ABB RobotStudio station: estacion_lab1_nike_plano.rsstn

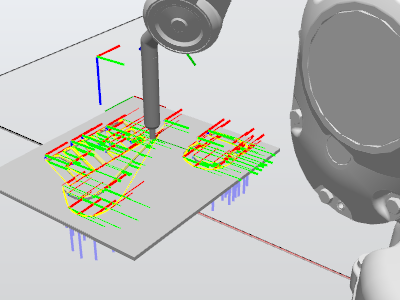
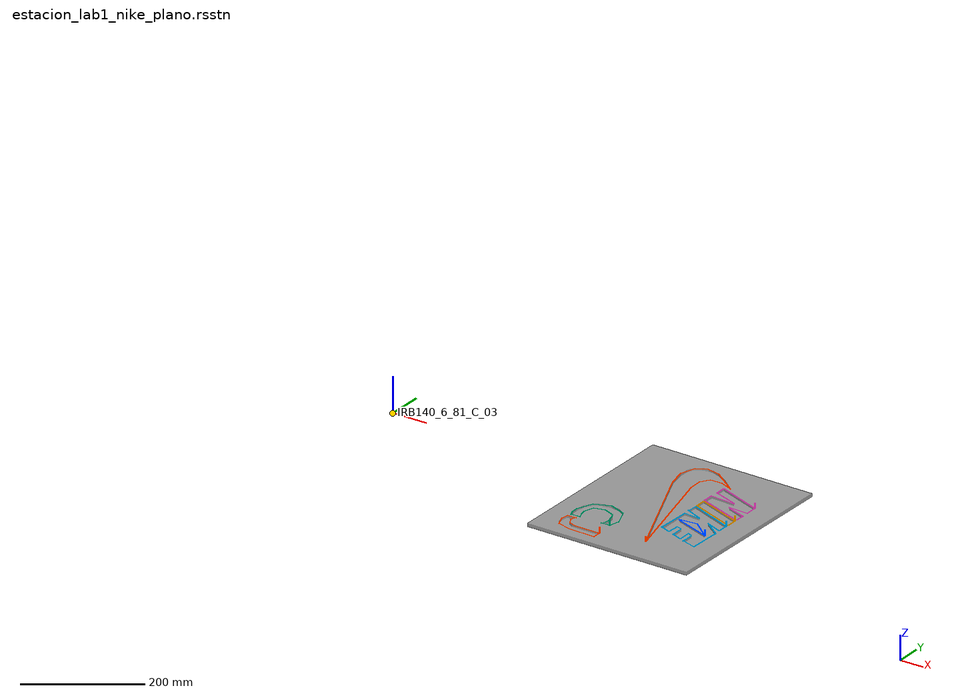
[picture v1: parts stored in the station drawn from their meshes, with robot base, taught points and paths (robot models come from the ABB library and are not in the file)]
Station estacion_lab1_nike_plano (saved by RobotStudio 24.1.10693.0)
Controller ControladorLab1
  mechanical unit ROB_1: IRB140_6_81_C_03, 6 joints, base frame (0, 0, 0) mm
Layout (positions relative to the parent item):
  - IRB140_6_81_C_03 [mechanism, from %ABB.RobotStudio.Models.IRB140%\IRB140_6_81_C_G_03.rslib] at (0, 0, 0) mm; joint values [-0.2293, 0.8636, 0.1936, 2.4826, 0.316, 2.0103] (rad or m)
  - Silueta_nike_nombres [part] at (550, 0, 0) mm, rotated rx 0 ry 0 rz -90 deg, size 349.5 x 310.3 x 6 mm
  - ToolLab1 [mechanism] at (562.41, -118.55, 208.97) mm, rotated rx -135 ry 0 rz -87.52 deg
      TCP ToolLab1 at (0.11, 120.32, 166.73) mm, rotated rx -45 ry 0 rz 0 deg
      links: HerramientaMarcadorEnsamblada v1
Attachment: ToolLab1 is attached to IRB140_6_81_C_03 / Link6
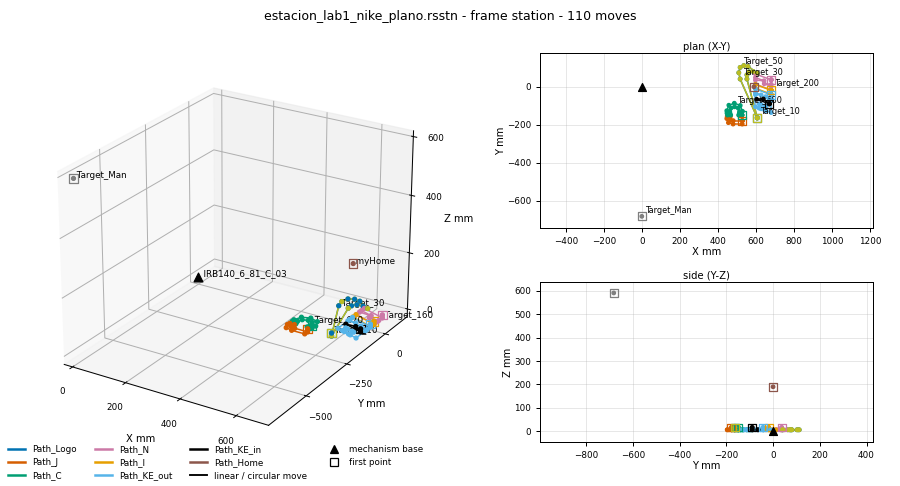
[picture p0: tool path of estacion_lab1_nike_plano.rsstn in frame station, 110 of 110 moves have a stored position in this frame; points joined in program order, loops and branches not executed]
Targets, tools, work objects and paths stored in the station, written as RAPID:
! task T_ROB1
MODULE CalibData
  PERS tooldata ToolLab1:=[TRUE,[[0.111,120.323,166.727],[0.923879533,-0.382683432,0,0]],[1,[0,0,1],[1,0,0,0],0,0,0]];
  TASK PERS wobjdata Workobject_1:=[FALSE,TRUE,"",[[722.891,-215.257,6],[0,0,1,0]],[[0,0,0],[1,0,0,0]]];
ENDMODULE

! task T_ROB1
MODULE Module1
  CONST robtarget Target_10:=[[115.3493902,51.778117998,-10],[0.69165817,0,0,-0.722225017],[0,0,0,0],[9E+09,9E+09,9E+09,9E+09,9E+09,9E+09]];
  CONST robtarget Target_20:=[[115.3493902,51.778117998,0],[0.69165817,0,0,-0.722225017],[0,0,0,0],[9E+09,9E+09,9E+09,9E+09,9E+09,9E+09]];
  CONST robtarget Target_30:=[[205.483730587,256.22918847,0],[0.69165817,0,0,-0.722225017],[0,0,0,0],[9E+09,9E+09,9E+09,9E+09,9E+09,9E+09]];
  CONST robtarget Target_40:=[[212.583843163,289.281706109,0],[0.69165817,0,0,-0.722225017],[0,0,0,0],[9E+09,9E+09,9E+09,9E+09,9E+09,9E+09]];
  CONST robtarget Target_50:=[[205.483730587,317.417949705,0],[0.69165817,0,0,-0.722225017],[0,0,0,0],[9E+09,9E+09,9E+09,9E+09,9E+09,9E+09]];
  CONST robtarget Target_60:=[[186.065561002,327.253449307,0],[0.69165817,0,0,-0.722225017],[0,0,0,0],[9E+09,9E+09,9E+09,9E+09,9E+09,9E+09]];
  CONST robtarget Target_70:=[[164.044058996,322.576768388,0],[0.69165817,0,0,-0.722225017],[0,0,0,0],[9E+09,9E+09,9E+09,9E+09,9E+09,9E+09]];
  CONST robtarget Target_80:=[[115.3493902,287.739568507,0],[0.69165817,0,0,-0.722225017],[0,0,0,0],[9E+09,9E+09,9E+09,9E+09,9E+09,9E+09]];
  CONST robtarget Target_90:=[[137.113893268,295.786272701,0],[0.69165817,0,0,-0.722225017],[0,0,0,0],[9E+09,9E+09,9E+09,9E+09,9E+09,9E+09]];
  CONST robtarget Target_100:=[[159.309752186,294.100202202,0],[0.69165817,0,0,-0.722225017],[0,0,0,0],[9E+09,9E+09,9E+09,9E+09,9E+09,9E+09]];
  CONST robtarget Target_110:=[[169.98114276,278.010063881,0],[0.69165817,0,0,-0.722225017],[0,0,0,0],[9E+09,9E+09,9E+09,9E+09,9E+09,9E+09]];
  CONST robtarget Target_120:=[[169.942954093,256.22918847,0],[0.69165817,0,0,-0.722225017],[0,0,0,0],[9E+09,9E+09,9E+09,9E+09,9E+09,9E+09]];
  CONST robtarget Target_130:=[[115.3493902,51.778117998,0],[0.69165817,0,0,-0.722225017],[0,0,0,0],[9E+09,9E+09,9E+09,9E+09,9E+09,9E+09]];
  CONST robtarget Target_140:=[[115.3493902,51.778117998,-10],[0.69165817,0,0,-0.722225017],[0,0,0,0],[9E+09,9E+09,9E+09,9E+09,9E+09,9E+09]];
  CONST robtarget Target_820:=[[194.456890225,37.1750385,-10],[0.69165817,0,0,-0.722225017],[0,0,0,0],[9E+09,9E+09,9E+09,9E+09,9E+09,9E+09]];
  CONST robtarget Target_830:=[[194.456890225,37.1750385,0],[0.69165817,0,0,-0.722225017],[0,0,0,0],[9E+09,9E+09,9E+09,9E+09,9E+09,9E+09]];
  CONST robtarget Target_840:=[[194.456890225,19.215854827,0],[0.69165817,0,0,-0.722225017],[0,0,0,0],[9E+09,9E+09,9E+09,9E+09,9E+09,9E+09]];
  CONST robtarget Target_850:=[[242.694367034,19.215854827,0],[0.69165817,0,0,-0.722225017],[0,0,0,0],[9E+09,9E+09,9E+09,9E+09,9E+09,9E+09]];
  CONST robtarget Target_860:=[[267.332585958,26.674110857,0],[0.69165817,0,0,-0.722225017],[0,0,0,0],[9E+09,9E+09,9E+09,9E+09,9E+09,9E+09]];
  CONST robtarget Target_870:=[[275.866908778,48.232552415,0],[0.69165817,0,0,-0.722225017],[0,0,0,0],[9E+09,9E+09,9E+09,9E+09,9E+09,9E+09]];
  CONST robtarget Target_880:=[[273.640563695,59.883758352,0],[0.69165817,0,0,-0.722225017],[0,0,0,0],[9E+09,9E+09,9E+09,9E+09,9E+09,9E+09]];
  CONST robtarget Target_890:=[[256.794552563,59.883758352,0],[0.69165817,0,0,-0.722225017],[0,0,0,0],[9E+09,9E+09,9E+09,9E+09,9E+09,9E+09]];
  CONST robtarget Target_900:=[[260.282493194,49.494147962,0],[0.69165817,0,0,-0.722225017],[0,0,0,0],[9E+09,9E+09,9E+09,9E+09,9E+09,9E+09]];
  CONST robtarget Target_910:=[[255.699932897,40.254815866,0],[0.69165817,0,0,-0.722225017],[0,0,0,0],[9E+09,9E+09,9E+09,9E+09,9E+09,9E+09]];
  CONST robtarget Target_920:=[[241.952252006,37.1750385,0],[0.69165817,0,0,-0.722225017],[0,0,0,0],[9E+09,9E+09,9E+09,9E+09,9E+09,9E+09]];
  CONST robtarget Target_930:=[[194.456890225,37.1750385,0],[0.69165817,0,0,-0.722225017],[0,0,0,0],[9E+09,9E+09,9E+09,9E+09,9E+09,9E+09]];
  CONST robtarget Target_940:=[[194.456890225,37.1750385,-10],[0.69165817,0,0,-0.722225017],[0,0,0,0],[9E+09,9E+09,9E+09,9E+09,9E+09,9E+09]];
  CONST robtarget Target_620:=[[196.015331784,66.562793602,-10],[0.69165817,0,0,-0.722225017],[0,0,0,0],[9E+09,9E+09,9E+09,9E+09,9E+09,9E+09]];
  CONST robtarget Target_630:=[[196.015331784,66.562793602,0],[0.69165817,0,0,-0.722225017],[0,0,0,0],[9E+09,9E+09,9E+09,9E+09,9E+09,9E+09]];
  CONST robtarget Target_640:=[[213.380823435,66.562793602,0],[0.69165817,0,0,-0.722225017],[0,0,0,0],[9E+09,9E+09,9E+09,9E+09,9E+09,9E+09]];
  CONST robtarget Target_650:=[[209.818671301,75.134222174,0],[0.69165817,0,0,-0.722225017],[0,0,0,0],[9E+09,9E+09,9E+09,9E+09,9E+09,9E+09]];
  CONST robtarget Target_660:=[[208.631287257,84.818823287,0],[0.69165817,0,0,-0.722225017],[0,0,0,0],[9E+09,9E+09,9E+09,9E+09,9E+09,9E+09]];
  CONST robtarget Target_670:=[[215.718485773,103.03774722,0],[0.69165817,0,0,-0.722225017],[0,0,0,0],[9E+09,9E+09,9E+09,9E+09,9E+09,9E+09]];
  CONST robtarget Target_680:=[[234.902159242,109.97652273,0],[0.69165817,0,0,-0.722225017],[0,0,0,0],[9E+09,9E+09,9E+09,9E+09,9E+09,9E+09]];
  CONST robtarget Target_690:=[[253.380823435,103.445910485,0],[0.69165817,0,0,-0.722225017],[0,0,0,0],[9E+09,9E+09,9E+09,9E+09,9E+09,9E+09]];
  CONST robtarget Target_700:=[[260.282493194,85.857784326,0],[0.69165817,0,0,-0.722225017],[0,0,0,0],[9E+09,9E+09,9E+09,9E+09,9E+09,9E+09]];
  CONST robtarget Target_710:=[[259.002344771,75.765019947,0],[0.69165817,0,0,-0.722225017],[0,0,0,0],[9E+09,9E+09,9E+09,9E+09,9E+09,9E+09]];
  CONST robtarget Target_720:=[[255.161899502,66.562793602,0],[0.69165817,0,0,-0.722225017],[0,0,0,0],[9E+09,9E+09,9E+09,9E+09,9E+09,9E+09]];
  CONST robtarget Target_730:=[[271.636853119,66.562793602,0],[0.69165817,0,0,-0.722225017],[0,0,0,0],[9E+09,9E+09,9E+09,9E+09,9E+09,9E+09]];
  CONST robtarget Target_740:=[[274.809394863,76.655557981,0],[0.69165817,0,0,-0.722225017],[0,0,0,0],[9E+09,9E+09,9E+09,9E+09,9E+09,9E+09]];
  CONST robtarget Target_750:=[[275.866908778,89.41993646,0],[0.69165817,0,0,-0.722225017],[0,0,0,0],[9E+09,9E+09,9E+09,9E+09,9E+09,9E+09]];
  CONST robtarget Target_760:=[[265.032029372,118.362422545,0],[0.69165817,0,0,-0.722225017],[0,0,0,0],[9E+09,9E+09,9E+09,9E+09,9E+09,9E+09]];
  CONST robtarget Target_770:=[[236.163754789,128.90045594,0],[0.69165817,0,0,-0.722225017],[0,0,0,0],[9E+09,9E+09,9E+09,9E+09,9E+09,9E+09]];
  CONST robtarget Target_780:=[[205.032029372,117.063721246,0],[0.69165817,0,0,-0.722225017],[0,0,0,0],[9E+09,9E+09,9E+09,9E+09,9E+09,9E+09]];
  CONST robtarget Target_790:=[[193.121083175,86.303053343,0],[0.69165817,0,0,-0.722225017],[0,0,0,0],[9E+09,9E+09,9E+09,9E+09,9E+09,9E+09]];
  CONST robtarget Target_800:=[[196.015331784,66.562793602,0],[0.69165817,0,0,-0.722225017],[0,0,0,0],[9E+09,9E+09,9E+09,9E+09,9E+09,9E+09]];
  CONST robtarget Target_810:=[[196.015331784,66.562793602,-10],[0.69165817,0,0,-0.722225017],[0,0,0,0],[9E+09,9E+09,9E+09,9E+09,9E+09,9E+09]];
  CONST robtarget Target_150:=[[42.139334196,252.185341465,-10],[0.69165817,0,0,-0.722225017],[0,0,0,0],[9E+09,9E+09,9E+09,9E+09,9E+09,9E+09]];
  CONST robtarget Target_160:=[[42.139334196,252.185341465,0],[0.69165817,0,0,-0.722225017],[0,0,0,0],[9E+09,9E+09,9E+09,9E+09,9E+09,9E+09]];
  CONST robtarget Target_170:=[[42.139334196,228.631408424,0],[0.69165817,0,0,-0.722225017],[0,0,0,0],[9E+09,9E+09,9E+09,9E+09,9E+09,9E+09]];
  CONST robtarget Target_180:=[[78.791441846,231.421966019,0],[0.69165817,0,0,-0.722225017],[0,0,0,0],[9E+09,9E+09,9E+09,9E+09,9E+09,9E+09]];
  CONST robtarget Target_190:=[[42.139334196,217.406656484,0],[0.69165817,0,0,-0.722225017],[0,0,0,0],[9E+09,9E+09,9E+09,9E+09,9E+09,9E+09]];
  CONST robtarget Target_200:=[[42.139334196,198.709287388,0],[0.69165817,0,0,-0.722225017],[0,0,0,0],[9E+09,9E+09,9E+09,9E+09,9E+09,9E+09]];
  CONST robtarget Target_210:=[[125.092149675,229.242650118,0],[0.69165817,0,0,-0.722225017],[0,0,0,0],[9E+09,9E+09,9E+09,9E+09,9E+09,9E+09]];
  CONST robtarget Target_220:=[[125.092149675,250.145759986,0],[0.69165817,0,0,-0.722225017],[0,0,0,0],[9E+09,9E+09,9E+09,9E+09,9E+09,9E+09]];
  CONST robtarget Target_230:=[[79.933561376,247.245410935,0],[0.69165817,0,0,-0.722225017],[0,0,0,0],[9E+09,9E+09,9E+09,9E+09,9E+09,9E+09]];
  CONST robtarget Target_240:=[[125.092149675,263.867433334,0],[0.69165817,0,0,-0.722225017],[0,0,0,0],[9E+09,9E+09,9E+09,9E+09,9E+09,9E+09]];
  CONST robtarget Target_250:=[[125.092149675,282.718704196,0],[0.69165817,0,0,-0.722225017],[0,0,0,0],[9E+09,9E+09,9E+09,9E+09,9E+09,9E+09]];
  CONST robtarget Target_260:=[[42.139334196,252.185341465,0],[0.69165817,0,0,-0.722225017],[0,0,0,0],[9E+09,9E+09,9E+09,9E+09,9E+09,9E+09]];
  CONST robtarget Target_270:=[[42.139334196,252.185341465,-10],[0.69165817,0,0,-0.722225017],[0,0,0,0],[9E+09,9E+09,9E+09,9E+09,9E+09,9E+09]];
  CONST robtarget Target_280:=[[42.139334196,196.560480665,-10],[0.69165817,0,0,-0.722225017],[0,0,0,0],[9E+09,9E+09,9E+09,9E+09,9E+09,9E+09]];
  CONST robtarget Target_290:=[[42.139334196,196.560480665,0],[0.69165817,0,0,-0.722225017],[0,0,0,0],[9E+09,9E+09,9E+09,9E+09,9E+09,9E+09]];
  CONST robtarget Target_300:=[[42.139334196,176.310975913,0],[0.69165817,0,0,-0.722225017],[0,0,0,0],[9E+09,9E+09,9E+09,9E+09,9E+09,9E+09]];
  CONST robtarget Target_310:=[[125.092149675,207.54980264,0],[0.69165817,0,0,-0.722225017],[0,0,0,0],[9E+09,9E+09,9E+09,9E+09,9E+09,9E+09]];
  CONST robtarget Target_320:=[[125.092149675,227.799307392,0],[0.69165817,0,0,-0.722225017],[0,0,0,0],[9E+09,9E+09,9E+09,9E+09,9E+09,9E+09]];
  CONST robtarget Target_330:=[[42.139334196,196.560480665,0],[0.69165817,0,0,-0.722225017],[0,0,0,0],[9E+09,9E+09,9E+09,9E+09,9E+09,9E+09]];
  CONST robtarget Target_340:=[[42.139334196,196.560480665,-10],[0.69165817,0,0,-0.722225017],[0,0,0,0],[9E+09,9E+09,9E+09,9E+09,9E+09,9E+09]];
  CONST robtarget Target_350:=[[42.139334196,172.506326672,-10],[0.69165817,0,0,-0.722225017],[0,0,0,0],[9E+09,9E+09,9E+09,9E+09,9E+09,9E+09]];
  CONST robtarget Target_360:=[[42.139334196,172.506326672,0],[0.69165817,0,0,-0.722225017],[0,0,0,0],[9E+09,9E+09,9E+09,9E+09,9E+09,9E+09]];
  CONST robtarget Target_370:=[[42.139334196,151.881719507,0],[0.69165817,0,0,-0.722225017],[0,0,0,0],[9E+09,9E+09,9E+09,9E+09,9E+09,9E+09]];
  CONST robtarget Target_380:=[[71.552108332,163.412354314,0],[0.69165817,0,0,-0.722225017],[0,0,0,0],[9E+09,9E+09,9E+09,9E+09,9E+09,9E+09]];
  CONST robtarget Target_390:=[[42.139334196,141.525904472,0],[0.69165817,0,0,-0.722225017],[0,0,0,0],[9E+09,9E+09,9E+09,9E+09,9E+09,9E+09]];
  CONST robtarget Target_400:=[[42.139334196,79.739107583,0],[0.69165817,0,0,-0.722225017],[0,0,0,0],[9E+09,9E+09,9E+09,9E+09,9E+09,9E+09]];
  CONST robtarget Target_410:=[[68.644796093,89.495266886,0],[0.69165817,0,0,-0.722225017],[0,0,0,0],[9E+09,9E+09,9E+09,9E+09,9E+09,9E+09]];
  CONST robtarget Target_420:=[[68.644796093,112.068396757,0],[0.69165817,0,0,-0.722225017],[0,0,0,0],[9E+09,9E+09,9E+09,9E+09,9E+09,9E+09]];
  CONST robtarget Target_430:=[[76.609476409,115.000044968,0],[0.69165817,0,0,-0.722225017],[0,0,0,0],[9E+09,9E+09,9E+09,9E+09,9E+09,9E+09]];
  CONST robtarget Target_440:=[[76.609476409,92.426915098,0],[0.69165817,0,0,-0.722225017],[0,0,0,0],[9E+09,9E+09,9E+09,9E+09,9E+09,9E+09]];
  CONST robtarget Target_450:=[[95.783017195,99.484332887,0],[0.69165817,0,0,-0.722225017],[0,0,0,0],[9E+09,9E+09,9E+09,9E+09,9E+09,9E+09]];
  CONST robtarget Target_460:=[[95.783017195,122.057462758,0],[0.69165817,0,0,-0.722225017],[0,0,0,0],[9E+09,9E+09,9E+09,9E+09,9E+09,9E+09]];
  CONST robtarget Target_470:=[[105.984433721,125.812411271,0],[0.69165817,0,0,-0.722225017],[0,0,0,0],[9E+09,9E+09,9E+09,9E+09,9E+09,9E+09]];
  CONST robtarget Target_480:=[[105.984433721,103.2392814,0],[0.69165817,0,0,-0.722225017],[0,0,0,0],[9E+09,9E+09,9E+09,9E+09,9E+09,9E+09]];
  CONST robtarget Target_490:=[[125.092149675,110.272470314,0],[0.69165817,0,0,-0.722225017],[0,0,0,0],[9E+09,9E+09,9E+09,9E+09,9E+09,9E+09]];
  CONST robtarget Target_500:=[[125.092149675,174.029241077,0],[0.69165817,0,0,-0.722225017],[0,0,0,0],[9E+09,9E+09,9E+09,9E+09,9E+09,9E+09]];
  CONST robtarget Target_510:=[[95.103567547,172.645188801,0],[0.69165817,0,0,-0.722225017],[0,0,0,0],[9E+09,9E+09,9E+09,9E+09,9E+09,9E+09]];
  CONST robtarget Target_520:=[[125.092149675,184.401556537,0],[0.69165817,0,0,-0.722225017],[0,0,0,0],[9E+09,9E+09,9E+09,9E+09,9E+09,9E+09]];
  CONST robtarget Target_530:=[[125.092149675,204.226450296,0],[0.69165817,0,0,-0.722225017],[0,0,0,0],[9E+09,9E+09,9E+09,9E+09,9E+09,9E+09]];
  CONST robtarget Target_540:=[[42.139334196,172.506326672,0],[0.69165817,0,0,-0.722225017],[0,0,0,0],[9E+09,9E+09,9E+09,9E+09,9E+09,9E+09]];
  CONST robtarget Target_550:=[[42.139334196,172.506326672,-10],[0.69165817,0,0,-0.722225017],[0,0,0,0],[9E+09,9E+09,9E+09,9E+09,9E+09,9E+09]];
  CONST robtarget Target_560:=[[51.878020694,125.812411271,-10],[0.69165817,0,0,-0.722225017],[0,0,0,0],[9E+09,9E+09,9E+09,9E+09,9E+09,9E+09]];
  CONST robtarget Target_570:=[[51.878020694,125.812411271,0],[0.69165817,0,0,-0.722225017],[0,0,0,0],[9E+09,9E+09,9E+09,9E+09,9E+09,9E+09]];
  CONST robtarget Target_580:=[[83.615741936,151.339072267,0],[0.69165817,0,0,-0.722225017],[0,0,0,0],[9E+09,9E+09,9E+09,9E+09,9E+09,9E+09]];
  CONST robtarget Target_590:=[[118.70894586,149.733785216,0],[0.69165817,0,0,-0.722225017],[0,0,0,0],[9E+09,9E+09,9E+09,9E+09,9E+09,9E+09]];
  CONST robtarget Target_600:=[[51.878020694,125.812411271,0],[0.69165817,0,0,-0.722225017],[0,0,0,0],[9E+09,9E+09,9E+09,9E+09,9E+09,9E+09]];
  CONST robtarget Target_610:=[[51.878020694,125.812411271,-10],[0.69165817,0,0,-0.722225017],[0,0,0,0],[9E+09,9E+09,9E+09,9E+09,9E+09,9E+09]];
  CONST robtarget myHome:=[[132.890790113,215.256892578,-184.00006578],[0.691638553,0.000000186,-0.000000501,-0.722243803],[-1,0,2,0],[9E+09,9E+09,9E+09,9E+09,9E+09,9E+09]];
  CONST robtarget Target_Man:=[[723.002,-466.47,-585.677],[0.923879532,0.382683433,0,0],[-2,0,-2,0],[9E+09,9E+09,9E+09,9E+09,9E+09,9E+09]];
  PROC Path_Logo()
    MoveL Target_10,v200,z10,ToolLab1\WObj:=Workobject_1;
    MoveL Target_20,v200,z10,ToolLab1\WObj:=Workobject_1;
    MoveL Target_30,v200,z10,ToolLab1\WObj:=Workobject_1;
    MoveL Target_40,v200,z10,ToolLab1\WObj:=Workobject_1;
    MoveL Target_50,v200,z10,ToolLab1\WObj:=Workobject_1;
    MoveL Target_60,v200,z10,ToolLab1\WObj:=Workobject_1;
    MoveL Target_70,v200,z10,ToolLab1\WObj:=Workobject_1;
    MoveL Target_80,v200,z10,ToolLab1\WObj:=Workobject_1;
    MoveL Target_90,v200,z10,ToolLab1\WObj:=Workobject_1;
    MoveL Target_100,v200,z10,ToolLab1\WObj:=Workobject_1;
    MoveL Target_110,v200,z10,ToolLab1\WObj:=Workobject_1;
    MoveL Target_120,v200,z10,ToolLab1\WObj:=Workobject_1;
    MoveL Target_130,v200,z10,ToolLab1\WObj:=Workobject_1;
    MoveL Target_140,v200,z10,ToolLab1\WObj:=Workobject_1;
  ENDPROC
  PROC main()
    SetDO DO_01,1;
    Logo;
    SetDO DO_01,0;
    SetDO DO_02,1;
    Path_Home;
    Path_Man;
    SetDO DO_02,0;
  ENDPROC
  PROC Logo()
    Path_Home;
    Path_Logo;
    Path_N;
    Path_I;
    Path_KE_out;
    Path_KE_in;
    Path_C;
    Path_J;
    Path_Home;
  ENDPROC
  PROC Path_J()
    MoveL Target_820,v200,z10,ToolLab1\WObj:=Workobject_1;
    MoveL Target_830,v200,z10,ToolLab1\WObj:=Workobject_1;
    MoveL Target_840,v200,z10,ToolLab1\WObj:=Workobject_1;
    MoveL Target_850,v200,z10,ToolLab1\WObj:=Workobject_1;
    MoveL Target_860,v200,z10,ToolLab1\WObj:=Workobject_1;
    MoveL Target_870,v200,z10,ToolLab1\WObj:=Workobject_1;
    MoveL Target_880,v200,z10,ToolLab1\WObj:=Workobject_1;
    MoveL Target_890,v200,z10,ToolLab1\WObj:=Workobject_1;
    MoveL Target_900,v200,z10,ToolLab1\WObj:=Workobject_1;
    MoveL Target_910,v200,z10,ToolLab1\WObj:=Workobject_1;
    MoveL Target_920,v200,z10,ToolLab1\WObj:=Workobject_1;
    MoveL Target_930,v200,z10,ToolLab1\WObj:=Workobject_1;
    MoveL Target_940,v200,z10,ToolLab1\WObj:=Workobject_1;
  ENDPROC
  PROC Path_C()
    MoveL Target_620,v200,z10,ToolLab1\WObj:=Workobject_1;
    MoveL Target_630,v200,z10,ToolLab1\WObj:=Workobject_1;
    MoveL Target_640,v200,z10,ToolLab1\WObj:=Workobject_1;
    MoveL Target_650,v200,z10,ToolLab1\WObj:=Workobject_1;
    MoveL Target_660,v200,z10,ToolLab1\WObj:=Workobject_1;
    MoveL Target_670,v200,z10,ToolLab1\WObj:=Workobject_1;
    MoveL Target_680,v200,z10,ToolLab1\WObj:=Workobject_1;
    MoveL Target_690,v200,z10,ToolLab1\WObj:=Workobject_1;
    MoveL Target_700,v200,z10,ToolLab1\WObj:=Workobject_1;
    MoveL Target_710,v200,z10,ToolLab1\WObj:=Workobject_1;
    MoveL Target_720,v200,z10,ToolLab1\WObj:=Workobject_1;
    MoveL Target_730,v200,z10,ToolLab1\WObj:=Workobject_1;
    MoveL Target_740,v200,z10,ToolLab1\WObj:=Workobject_1;
    MoveL Target_750,v200,z10,ToolLab1\WObj:=Workobject_1;
    MoveL Target_760,v200,z10,ToolLab1\WObj:=Workobject_1;
    MoveL Target_770,v200,z10,ToolLab1\WObj:=Workobject_1;
    MoveL Target_780,v200,z10,ToolLab1\WObj:=Workobject_1;
    MoveL Target_790,v200,z10,ToolLab1\WObj:=Workobject_1;
    MoveL Target_800,v200,z10,ToolLab1\WObj:=Workobject_1;
    MoveL Target_810,v200,z10,ToolLab1\WObj:=Workobject_1;
  ENDPROC
  PROC Path_N()
    MoveL Target_150,v200,z10,ToolLab1\WObj:=Workobject_1;
    MoveL Target_160,v200,z10,ToolLab1\WObj:=Workobject_1;
    MoveL Target_170,v200,z10,ToolLab1\WObj:=Workobject_1;
    MoveL Target_180,v200,z10,ToolLab1\WObj:=Workobject_1;
    MoveL Target_190,v200,z10,ToolLab1\WObj:=Workobject_1;
    MoveL Target_200,v200,z10,ToolLab1\WObj:=Workobject_1;
    MoveL Target_210,v200,z10,ToolLab1\WObj:=Workobject_1;
    MoveL Target_220,v200,z10,ToolLab1\WObj:=Workobject_1;
    MoveL Target_230,v200,z10,ToolLab1\WObj:=Workobject_1;
    MoveL Target_240,v200,z10,ToolLab1\WObj:=Workobject_1;
    MoveL Target_250,v200,z10,ToolLab1\WObj:=Workobject_1;
    MoveL Target_260,v200,z10,ToolLab1\WObj:=Workobject_1;
    MoveL Target_270,v200,z10,ToolLab1\WObj:=Workobject_1;
  ENDPROC
  PROC Path_I()
    MoveL Target_280,v200,z10,ToolLab1\WObj:=Workobject_1;
    MoveL Target_290,v200,z10,ToolLab1\WObj:=Workobject_1;
    MoveL Target_300,v200,z10,ToolLab1\WObj:=Workobject_1;
    MoveL Target_310,v200,z10,ToolLab1\WObj:=Workobject_1;
    MoveL Target_320,v200,z10,ToolLab1\WObj:=Workobject_1;
    MoveL Target_330,v200,z10,ToolLab1\WObj:=Workobject_1;
    MoveL Target_340,v200,z10,ToolLab1\WObj:=Workobject_1;
  ENDPROC
  PROC Path_KE_out()
    MoveL Target_350,v200,z10,ToolLab1\WObj:=Workobject_1;
    MoveL Target_360,v200,z10,ToolLab1\WObj:=Workobject_1;
    MoveL Target_370,v200,z10,ToolLab1\WObj:=Workobject_1;
    MoveL Target_380,v200,z10,ToolLab1\WObj:=Workobject_1;
    MoveL Target_390,v200,z10,ToolLab1\WObj:=Workobject_1;
    MoveL Target_400,v200,z10,ToolLab1\WObj:=Workobject_1;
    MoveL Target_410,v200,z10,ToolLab1\WObj:=Workobject_1;
    MoveL Target_420,v200,z10,ToolLab1\WObj:=Workobject_1;
    MoveL Target_430,v200,z10,ToolLab1\WObj:=Workobject_1;
    MoveL Target_440,v200,z10,ToolLab1\WObj:=Workobject_1;
    MoveL Target_450,v200,z10,ToolLab1\WObj:=Workobject_1;
    MoveL Target_460,v200,z10,ToolLab1\WObj:=Workobject_1;
    MoveL Target_470,v200,z10,ToolLab1\WObj:=Workobject_1;
    MoveL Target_480,v200,z10,ToolLab1\WObj:=Workobject_1;
    MoveL Target_490,v200,z10,ToolLab1\WObj:=Workobject_1;
    MoveL Target_500,v200,z10,ToolLab1\WObj:=Workobject_1;
    MoveL Target_510,v200,z10,ToolLab1\WObj:=Workobject_1;
    MoveL Target_520,v200,z10,ToolLab1\WObj:=Workobject_1;
    MoveL Target_530,v200,z10,ToolLab1\WObj:=Workobject_1;
    MoveL Target_540,v200,z10,ToolLab1\WObj:=Workobject_1;
    MoveL Target_550,v200,z10,ToolLab1\WObj:=Workobject_1;
  ENDPROC
  PROC Path_KE_in()
    MoveL Target_560,v200,z10,ToolLab1\WObj:=Workobject_1;
    MoveL Target_570,v200,z10,ToolLab1\WObj:=Workobject_1;
    MoveL Target_580,v200,z10,ToolLab1\WObj:=Workobject_1;
    MoveL Target_590,v200,z10,ToolLab1\WObj:=Workobject_1;
    MoveL Target_600,v200,z10,ToolLab1\WObj:=Workobject_1;
    MoveL Target_610,v200,z10,ToolLab1\WObj:=Workobject_1;
  ENDPROC
  PROC Path_Home()
    MoveJ myHome,v200,z10,ToolLab1\WObj:=Workobject_1;
  ENDPROC
  PROC Path_Man()
    MoveJ Target_Man,v200,z10,ToolLab1\WObj:=Workobject_1;
  ENDPROC
  PROC Path_10()
    MoveL Target_10,v200,z10,ToolLab1\WObj:=Workobject_1;
    MoveL Target_20,v200,z10,ToolLab1\WObj:=Workobject_1;
    MoveL Target_30,v200,z10,ToolLab1\WObj:=Workobject_1;
    MoveL Target_40,v200,z10,ToolLab1\WObj:=Workobject_1;
    MoveL Target_50,v200,z10,ToolLab1\WObj:=Workobject_1;
    MoveL Target_60,v200,z10,ToolLab1\WObj:=Workobject_1;
    MoveL Target_70,v200,z10,ToolLab1\WObj:=Workobject_1;
    MoveL Target_80,v200,z10,ToolLab1\WObj:=Workobject_1;
    MoveL Target_90,v200,z10,ToolLab1\WObj:=Workobject_1;
    MoveL Target_100,v200,z10,ToolLab1\WObj:=Workobject_1;
    MoveL Target_110,v200,z10,ToolLab1\WObj:=Workobject_1;
    MoveL Target_120,v200,z10,ToolLab1\WObj:=Workobject_1;
    MoveL Target_130,v200,z10,ToolLab1\WObj:=Workobject_1;
    MoveL Target_140,v200,z10,ToolLab1\WObj:=Workobject_1;
  ENDPROC
ENDMODULE

